// TIA Portal V21 export
DATA_BLOCK "Data_block_1"   // DB1
{ S7_Optimized_Access := 'TRUE' }
// stored: MemoryReserve 100
   VAR
      Variable3 : Bool;
      Variable4 : Int := 164;
   END_VAR
BEGIN
END_DATA_BLOCK
